// TIA Portal V17 export
// export: Created 2025-06-26T07:49:37.2389884Z, ExportSetting WithDefaults, DisplayName Totally Integrated Automation Portal, DisplayVersion V17 Update 8, DisplayName TIA Portal Openness, DisplayVersion V17 Update 8, DisplayName TIA Portal Version Control Interface, DisplayVersion V17, DisplayName STEP 7 Professional, DisplayVersion V17 Update 8, DisplayName STEP 7 Safety, DisplayVersion V17 Update 6, DisplayName WinCC Advanced, DisplayVersion V17 Update 8
FUNCTION_BLOCK "OilHeating"   // FB17, FBD
TITLE = Crankcase oil sump heating control
{ S7_Optimized_Access := 'TRUE' }
VERSION : 0.1
// stored: AutoNumber true, IsIECCheckEnabled false, IsRetainMemResEnabled false, MemoryReserve 100, SetENOAutomatically false, UDAEnableTagReadback false
   VAR_INPUT
      bEnable { ExternalAccessible := 'False'; ExternalVisible := 'False'; ExternalWritable := 'False'} : Bool;
      bReset { ExternalAccessible := 'False'; ExternalVisible := 'False'; ExternalWritable := 'False'} : Bool;   // 1 = reset manual modes
   END_VAR
   VAR
      sHeaterControl { ExternalAccessible := 'False'; ExternalVisible := 'False'; ExternalWritable := 'False'} : "fbOnOffRegulator";
      bHeating { ExternalAccessible := 'False'; ExternalVisible := 'False'; ExternalWritable := 'False'; S7_SetPoint := 'True'} : Bool;
      A5000 { ExternalAccessible := 'False'; ExternalVisible := 'False'; ExternalWritable := 'False'; S7_SetPoint := 'True'} : "fbDigitalAlarm";
      A5001 { ExternalAccessible := 'False'; ExternalVisible := 'False'; ExternalWritable := 'False'; S7_SetPoint := 'True'} : "fbDigitalAlarm";
   END_VAR
   VAR_TEMP
      fSetpoint : Real;
   END_VAR
BEGIN

REGION Network 1 (SCL): Setpoint selection
   // Heating setpoint selection
   #fSetpoint := MAX(IN1 := "DB_CurrentSetting".VariableSetting.OilHeatSetpoint_min, IN2 := "DB_Calc".Compressor.CrankcaseSaturationTemperature.fValue + "DB_Regulators".OilHeating.fOilSuperheat);
   // Heating setpoint limitation
   "DB_Regulators".OilHeating.Controller.fSetpoint := MIN(IN1:= #fSetpoint, IN2:= "DB_CurrentSetting".Fluid.Limits.T_OilTemperature_Critical - 15);
END_REGION

REGION Network 2: Regulator
   // Additional criteria for running: crankcase wall temperatures are not above limit
   // Use the alarms to set time delay & hysteresis to prevent frequent triggering
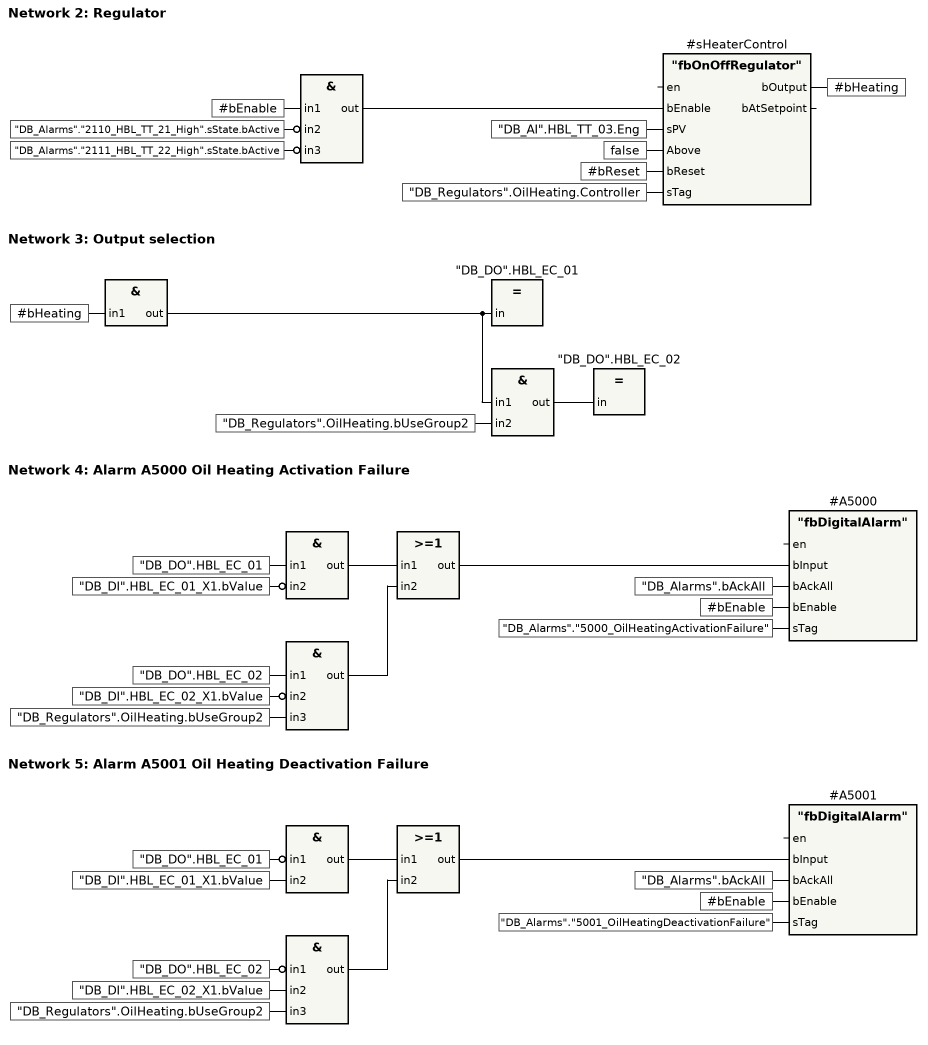
   #sHeaterControl(bEnable := #bEnable AND NOT "DB_Alarms"."2110_HBL_TT_21_High".sState.bActive AND NOT "DB_Alarms"."2111_HBL_TT_22_High".sState.bActive,   // "fbOnOffRegulator"
                   sPV := "DB_AI".HBL_TT_03.Eng,
                   Above := false,
                   bReset := #bReset,
                   sTag := "DB_Regulators".OilHeating.Controller,
                   bOutput => #bHeating);
END_REGION

REGION Network 3: Output selection
   // Selection of heater groups is manual for now. If programmatic selection is needed, change the code here :-)
   "DB_DO".HBL_EC_01 := #bHeating;
   "DB_DO".HBL_EC_02 := #bHeating AND "DB_Regulators".OilHeating.bUseGroup2;
END_REGION

REGION Network 4: Alarm A5000 Oil Heating Activation Failure
   #A5000(bInput := ("DB_DO".HBL_EC_01 AND NOT "DB_DI".HBL_EC_01_X1.bValue) OR ("DB_DO".HBL_EC_02 AND NOT "DB_DI".HBL_EC_02_X1.bValue AND "DB_Regulators".OilHeating.bUseGroup2),   // "fbDigitalAlarm"
          bAckAll := "DB_Alarms".bAckAll,
          bEnable := #bEnable,
          sTag := "DB_Alarms"."5000_OilHeatingActivationFailure");
END_REGION

REGION Network 5: Alarm A5001 Oil Heating Deactivation Failure
   #A5001(bInput := (NOT "DB_DO".HBL_EC_01 AND "DB_DI".HBL_EC_01_X1.bValue) OR (NOT "DB_DO".HBL_EC_02 AND "DB_DI".HBL_EC_02_X1.bValue AND "DB_Regulators".OilHeating.bUseGroup2),   // "fbDigitalAlarm"
          bAckAll := "DB_Alarms".bAckAll,
          bEnable := #bEnable,
          sTag := "DB_Alarms"."5001_OilHeatingDeactivationFailure");
END_REGION
END_FUNCTION_BLOCK
